INTERFACE I_PersistentEventStorage

METHOD StoreEvent
VAR_INPUT
	stEvent : ST_Event;
END_VAR
END_METHOD

END_INTERFACE

(* stored: Version 1.1.0.1, ProductVersion 3.1.4024.15
   Itf I_PersistentEventStorage: Id {6bcab42f-4f05-431e-b6ec-23cd3682557c}
   Method StoreEvent: Id {afe1e306-9117-4b72-ad49-6c0faf987f67} *)
